(* PLC project flow_sensor, Dassault Systèmes ControlBuild 2024x *)
(* stored: creationDateTime 2023-10-03T11:12:57-01:00 *)

(* This module simulates the behaviour of a flow sensor. The flow is measured in litre / min (use this module with the module flow_compute). *)
FUNCTION_BLOCK equipment_library.flow_sensor
  VAR_INPUT
    inputFlow : REAL := 0.0;
  END_VAR
  VAR_OUTPUT
    outputFlow : REAL := 0.0;
  END_VAR
  VAR
    unit : REAL := 0.0;
  END_VAR
  VAR CONSTANT
    flowPerHour : BOOL := true;
    flowPerMinute : BOOL := false;
  END_VAR
  VAR
    d_flow : BOOL := false;
    v_d_flow : REAL := 0.0;
  END_VAR


ACTION C_source_code:
/* -----------------------------------------------------------------	*/
/* Type : Model of Operative Behaviour					*/
/* Catégorie :   batch							*/
/* Author : Dassault Systemes						*/
/* Update date : June 2018							*/
/* -----------------------------------------------------------------	*/
/* This module simulates the behaviour of a flow sensor.		*/
/* The flow is measured in litre / min.					*/
/* This module should be used with the module flow_compute.		*/
/* ----------------------------------------------------------------	*/

if (flowPerHour) unit = 3600.0;
else if (flowPerMinute) unit = 60.0;
	else unit = 1.0;

if (!d_flow)
	outputFlow = (inputFlow / CLOCK_PERIOD * 1000000) * unit;
else
	outputFlow = v_d_flow;
END_ACTION
END_FUNCTION_BLOCK
